(* IEC 61131-3 sources: json/src/Types, 3 files *)

(* ---- IJsonProperty.st ---- *)
NAMESPACE Simatic.Ax.Json
    INTERFACE IJsonProperty EXTENDS IJsonObject
    END_INTERFACE
END_NAMESPACE

(* ---- DoubleInt.st ---- *)
USING Simatic.Ax.Conversion;
USING Simatic.Ax.Conversion;

NAMESPACE Simatic.Ax.Json.Properties
    CLASS DoubleInt EXTENDS JsonProperty
        VAR PUBLIC
            value : DINT;
        END_VAR

        METHOD PUBLIC OVERRIDE ToString : STRING
            ToString := THIS.ToStringHelper(Integer.ToString(value := value));
        END_METHOD
    END_CLASS
END_NAMESPACE

(* ---- JsonProperty.st ---- *)
USING System.Strings;

NAMESPACE Simatic.Ax.Json
    CLASS ABSTRACT JsonProperty IMPLEMENTS IJsonProperty
        VAR PUBLIC
            key : STRING;
        END_VAR

        VAR PROTECTED
            _next : IJsonProperty;
        END_VAR

        METHOD PUBLIC ABSTRACT ToString : STRING
        END_METHOD

        METHOD PUBLIC Serialize : BOOL
            VAR_INPUT
                t : ARRAY [*] OF BYTE;
            END_VAR
            ;
        END_METHOD

        METHOD PROTECTED ToStringHelper : STRING
            VAR_INPUT
                valueAsString : STRING;
            END_VAR
            VAR_TEMP
                _str : STRING;
            END_VAR
            _str := Concat('"', key, '"', ': "');
            _str := Concat(_str, valueAsString, '"');
            ToStringHelper := _str;
        END_METHOD
    END_CLASS
END_NAMESPACE
